FUNCTION_BLOCK FB_MathCalculation
VAR_INPUT
END_VAR
VAR_OUTPUT 
	bError : BOOL;
	ipResultMessage : I_TcMessage := fbResult;
END_VAR

VAR
	fbResult : FB_TcMessage;
(*	fbSource : FB_TcSourceInfo;	// optional *)
	
	hrLastInternalError : HRESULT;
	
	 {attribute 'hide'}
	bOwnTL : BOOL; // own trace level is set
	 {attribute 'hide'}
	eOwnTL : TcEventSeverity := TcEventSeverity.Critical;
END_VAR

// returns TRUE if succeeded
METHOD Addition : BOOL
VAR_INPUT
	nIn1 : UDINT;
	nIn2 : UDINT;
	nSum : REFERENCE TO UDINT;
END_VAR

VAR
	hr : HRESULT;
END_VAR
nSum := nIn1 + nIn2;

IF (nSum < nIn1) THEN // an overflow occurred
	bError := TRUE;

	IF NOT fbResult.EqualsToEventEntryEx(stOther:=TC_EVENTS.Win32EventClass.ERROR_ARITHMETIC_OVERFLOW) THEN
		hr := fbResult.CreateEx(TC_EVENTS.Win32EventClass.ERROR_ARITHMETIC_OVERFLOW, 0 ); //This uses dyn ressources and shouldn't be called cyclically.
		IF FAILED(hr) THEN
			hrLastInternalError := hr;
		END_IF
		
		IF fbResult.eSeverity >= eTraceLevel THEN
			hr := fbResult.Send(0);
			IF FAILED(hr) THEN
				hrLastInternalError := hr;
			END_IF
		END_IF 
	END_IF
	
ELSE
	Addition := TRUE;
	bError := FALSE;
	IF NOT fbResult.EqualsToEventEntryEx(stOther:=SUCCESS_EVENT) THEN
		hr := fbResult.CreateEx(SUCCESS_EVENT, 0 ); //This uses dyn ressources and shouldn't be called cyclically.
		IF FAILED(hr) THEN
			hrLastInternalError := hr;
		END_IF
	END_IF
	
END_IF
END_METHOD

// whether the event trace level is taken from the library default or not. This could be set via Online View too.
{attribute 'monitoring':='call'}
PROPERTY bTraceLevelDefault : BOOL
GET
bTraceLevelDefault := NOT bOwnTL;
END_GET
SET
bOwnTL := NOT bTraceLevelDefault;
END_SET
END_PROPERTY

// returns TRUE if succeeded
METHOD Division : BOOL
VAR_INPUT
	fDividend : LREAL;
	fDivisor  : LREAL;
	fQuotient : REFERENCE TO LREAL;
END_VAR

VAR
	hr : HRESULT;
END_VAR
IF (fDivisor = 0) THEN
	bError := TRUE;
	//adapt source name if required (default is ads symbol name)
	//fbSource.Clear();
	//fbSource.sName := 'Math Calculation';
	IF NOT fbResult.EqualsToEventEntryEx(stOther:=TC_EVENTS.CalculationEventClass.DivisionByZero) THEN
		hr := fbResult.CreateEx(TC_EVENTS.CalculationEventClass.DivisionByZero, 0 (*fbSource*) ); //This uses dyn ressources and shouldn't be called cyclically.
		IF FAILED(hr) THEN
			hrLastInternalError := hr;
		END_IF
		//set Arguments if required
		//fbResult.ipArguments.Clear().Add ...
		//set JSON attribute if required
		//fbResult.SetJsonAttribute('{"DivionByZero":1,"Divisor":0}');
		
		IF fbResult.eSeverity >= eTraceLevel THEN
			hr := fbResult.Send(0);
			IF FAILED(hr) THEN
				hrLastInternalError := hr;
			END_IF
		END_IF 
	END_IF
	
ELSE
	fQuotient := fDividend / fDivisor;
	Division := TRUE;
	bError := FALSE;
	IF NOT fbResult.EqualsToEventEntryEx(stOther:=SUCCESS_EVENT) THEN
		hr := fbResult.CreateEx(SUCCESS_EVENT, 0 (*fbSource*) ); //This uses dyn ressources and shouldn't be called cyclically.
		IF FAILED(hr) THEN
			hrLastInternalError := hr;
		END_IF
	END_IF
	
END_IF
END_METHOD

// current trace level for this FB. This could be set via Online View too. 
{attribute 'monitoring':='call'}
PROPERTY eTraceLevel : TcEventSeverity
GET
IF bOwnTL THEN
	eTraceLevel := eOwnTL;
ELSE
	eTraceLevel := GVL.eEventTraceLevel;
END_IF
END_GET
SET
bOwnTL := TRUE;
eOwnTL := eTraceLevel;
END_SET
END_PROPERTY

END_FUNCTION_BLOCK

(* stored: Version 1.1.0.1, ProductVersion 3.1.4022.10
   POU FB_MathCalculation: Id {f3553769-4f87-43e5-9171-428078be63d2}, SpecialFunc None
   Method Addition: Id {148727a5-02cd-4163-8e79-95a15c9851c8}
   Property bTraceLevelDefault: Id {ee6b29d3-e8c3-4031-b236-440c8959e66a}
   Get Get: Id {324ca596-f337-4258-a112-fb33c200676d}
   Set Set: Id {d5eef79d-4e5e-4499-849e-1421233d08b0}
   Method Division: Id {da0279bc-ff01-4b2a-b792-30ddd4c9187d}
   Property eTraceLevel: Id {ff84487f-e850-4269-a2de-648da5e8ea8c}
   Get Get: Id {feefb493-8041-4828-828b-d8af7ea1ed1b}
   Set Set: Id {e6d3034a-ec28-4113-8711-e467e0effe5b} *)
